Staubli VAL3: getConvFrame.pgx

public program getConvFrame(num x_nConvNum (dimensions=1), frame& x_fConveyor (dimensions=1), frame x_fRefFrame (dimensions=1), num& x_nError (dimensions=1))
begin
  // This program returns the position and orientation of the conveyor
  //  frame in reference to the frame x_fRefFrame.
  //
  // Input Param
  //  x_nConvNum : Conveyor number
  //  x_fRefFrame: Reference frame from which the coordinates of
  //                x_fConveyor should be returned.
  //
  // Output param
  //  x_fConveyor: Coordinates of the conveyor’s frame that have been
  //                taught during calibration.
  //  x_nError   : Error code
  //    0    --> No error
  //    14   --> Conveyor library not started, the frame cannot be computed.
  //
  //----------------------------------------------------------------
  //
  switch x_nConvNum
    case 0
      if cnv0:libExist("getConvFrame()")
        call cnv0:getConvFrame(x_fConveyor,x_fRefFrame,x_nError)
        if x_nError!=0
          call cnv0:getErrorMessage(sErrorMessage)
        endIf
      else
        nStatus=-1
      endIf
    break
    case 1
      if cnv1:libExist("getConvFrame()")
        call cnv1:getConvFrame(x_fConveyor,x_fRefFrame,x_nError)
        if x_nError!=0
          call cnv1:getErrorMessage(sErrorMessage)
        endIf
      else
        nStatus=-1
      endIf
    break
  endSwitch
end
